FUNCTION_BLOCK FIELDBUS_BYTE_TO_SIGNAL_SCALED (* Mirrors IN->OUT if Signal Valid, with scaling *)
  (* Standard: 61499-1; Description: Copyright (c) 2026 HR Agrartechnik GmbH This program and the accompanying materials are made available under the terms of the Eclipse Public License 2.0 which is available at https://www.eclipse.org/legal/epl-2.0/ SPDX-License-Identifier: EPL-2.0 *)
  (* Version 1.0, 2026-05-31, Franz Höpfinger, HR Agrartechnik GmbH *)
  PACKAGE logiBUS::signalprocessing::fieldbus;
  IMPORT signalprocessing::FIELDBUS_SIGNAL::NOT_AVAILABLE_B;
  IMPORT signalprocessing::FIELDBUS_SIGNAL::VALID_SIGNAL_B;
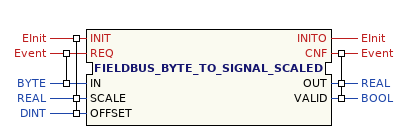
  EVENT_INPUT
    INIT : EInit WITH SCALE, OFFSET; (* Init Request *)
    REQ WITH IN; (* Normal Execution Request *)
  END_EVENT
  EVENT_OUTPUT
    INITO : EInit; (* Init Confirmation *)
    CNF WITH OUT, VALID; (* Execution Confirmation *)
  END_EVENT
  VAR_INPUT
    IN : BYTE := NOT_AVAILABLE_B; (* Input *)
    SCALE : REAL := REAL#1.0; (* Scaling factor *)
    OFFSET : DINT := DINT#0; (* Offset added after scaling *)
  END_VAR
  VAR_OUTPUT
    OUT : REAL := REAL#0.0; (* Output Scaled *)
    VALID : BOOL := FALSE; (* TRUE if Signal is VALID *)
  END_VAR
  EC_STATES
    INIT : INIT -> INITO;
    REQ : REQ -> CNF;
  END_STATES
  ALGORITHM INIT IN ST:

  END_ALGORITHM
  ALGORITHM REQ IN ST: (* Executed algorithm *)
IF (IN <= VALID_SIGNAL_B) THEN
	OUT := USINT_TO_REAL(BYTE_TO_USINT(IN)) * SCALE + DINT_TO_REAL(OFFSET);
	VALID := BOOL#TRUE;
ELSE
	OUT := REAL#0.0;
	VALID := BOOL#FALSE;
END_IF;
  END_ALGORITHM
END_FUNCTION_BLOCK
